Fanuc KAREL source: kt00611.KL

-- PROVISIONAL review KL for V770-1; original PC SHA256 159a9b763e06e91cad5b46409049abaf1e7e883049a8db3db05f4b6f4de2a66b
-- Incomplete behavior may be omitted. Consult companion uncertainty JSON. Do not deploy.
PROGRAM KT00611
%NOLOCKGROUP
VAR
  R1 : REAL
  R2 : REAL
  OUT : REAL
BEGIN
  -- UNRESOLVED_PC offsets 5-16; opcodes 2E,23
  -- UNRESOLVED_PC offsets 21-32; opcodes 2E,23
  -- UNRESOLVED_PC offsets 37-48; opcodes 2E,23
  -- UNRESOLVED_PC offsets 53-64; opcodes 2E,23
  -- UNRESOLVED_PC offsets 69-81; opcodes 21,23
  -- UNRESOLVED_PC offsets 86-90; opcodes 7F
END KT00611
